PROGRAM Gripper
VAR_INPUT
	closeGripperCommand : BOOL;
END_VAR
VAR
	closeGripperFromSimulink AT%I* : LREAL:=0;
	//closeGripperCommand		AT%I* : BOOL;				//True: opening, false: closing
	slider					AT%I* : BOOL;
	partGripped				AT%I* : BOOL;
	
	sliderToSimulink 		AT%Q* : LREAL:=0;
	partInGripperToSimulink AT%Q*  :LREAL:=0;
	
	driveEnable				AT%Q* : BOOL;
	driveVelocity 			AT%Q* : INT;
	
	state : CoreGripperControlState := CoreGripperControlState.Open;
	
	timer : TON;
	
	movementTime : TIME := T#1.0S;
	
END_VAR

CASE state OF 
		
	CoreGripperControlState.Opening:
		driveEnable:=1;
		driveVelocity:=-32767;
		timer(IN:=1);
		
		IF timer.Q THEN state := CoreGripperControlState.Open;
		END_IF
		
		IF closeGripperFromSimulink < 0.5 AND NOT closeGripperCommand THEN
			state := CoreGripperControlState.Closing;
			timer(in := 0, pt:= movementTime);
		END_IF
		
	CoreGripperControlState.Closing:
		driveEnable:=1;
		driveVelocity:=32767;
		timer(IN:=1);
		
		IF timer.Q THEN state := CoreGripperControlState.Closed;
		END_IF
		
		IF closeGripperFromSimulink > 0.5 OR  closeGripperCommand THEN
			state := CoreGripperControlState.Opening;
			timer(in := 0, pt:= movementTime);
		END_IF
		
		
	CoreGripperControlState.Open:	
		driveEnable:=0;
		driveVelocity:=0;

		IF closeGripperFromSimulink < 0.5 AND NOT closeGripperCommand THEN
			state := CoreGripperControlState.Closing;
			timer(in := 0, pt:= movementTime);
		END_IF
		
	CoreGripperControlState.Closed:	
		driveEnable:=0;
		driveVelocity:=0;
		
		IF closeGripperFromSimulink > 0.5 OR closeGripperCommand THEN
			state := CoreGripperControlState.Opening;
			timer(in := 0, pt:= movementTime);
		END_IF
		
END_CASE

sliderToSimulink:=BOOL_TO_LREAL(NOT(slider));
partInGripperToSimulink:=BOOL_TO_LREAL(NOT(partGripped));

END_PROGRAM

(* stored: Version 1.1.0.1, ProductVersion 3.1.4024.11
   POU Gripper: Id {914b4c40-8d67-4edc-a810-6f17709861da}, SpecialFunc None *)
